// Mitsubishi GX Works2 project: PLC- Group36   PLC: FX3G

// global labels: Global1
VAR_GLOBAL
  Start AT X007 : BOOL;
  M_Cream AT D1100 : INT;
END_VAR
VAR_GLOBAL CONSTANT
  Min_Cream : INT := 300;
END_VAR
VAR_GLOBAL
  M_Chocolate AT D1200 : INT;
END_VAR
VAR_GLOBAL CONSTANT
  Min_Chocolate : INT := 240;
END_VAR
VAR_GLOBAL
  M_Bisc AT D1300 : INT;
END_VAR
VAR_GLOBAL CONSTANT
  Min_Bisc : INT := 6;
END_VAR
VAR_GLOBAL
  Lamp_Start AT Y007 : BOOL;
  KJK AT Y005 : BOOL;
  Start2 AT X010 : BOOL;
  Start_Cream AT X011 : BOOL;
END_VAR
VAR_GLOBAL CONSTANT
  Less_Cream : INT := 300;
  Less_Bisc : INT := 6;
END_VAR
VAR_GLOBAL
  Start_Dipping AT X006 : BOOL;
  Analog_Input1 AT D8280 : INT;
  Save_analog1 AT D8201 : INT;
  SaveLampInput AT M1 : BOOL;
END_VAR
VAR_GLOBAL CONSTANT
  Min_Analog1 : INT := 6;
  Max_Analog1 : INT := 5;
  Less_ChocolateA : INT := 240;
  Less_ChocolateB : INT := 120;
END_VAR
VAR_GLOBAL
  Timer_Dipping AT TC10 : BOOL;
END_VAR
VAR_GLOBAL CONSTANT
  Time_Value : INT := 50;
END_VAR
VAR_GLOBAL
  Lamp_Dipping AT Y003 : BOOL;
END_VAR
VAR_GLOBAL CONSTANT
  Div_Analog1 : INT := 400;
END_VAR
VAR_GLOBAL
  Time_1 AT TS10 : BOOL;
  check AT X000 : BOOL;
  Input_Cream AT D1110 : INT;
  Input_Bisc AT D1310 : INT;
  Input_Chocolate AT D1210 : INT;
  Time_10 AT M10 : BOOL;
  Timer_Moving AT TC2 : BOOL;
  Time_Value2 AT K10 : INT;
  Time_2 AT TS2 : BOOL;
  Moving_Lamp0 AT Y000 : BOOL;
  Timer_Moving2 AT TC3 : BOOL;
  Time_Value3 AT K10 : INT;
  Time_3 AT TS3 : BOOL;
  Moving_Lamp1 AT Y001 : BOOL;
  Timer_Moving3 AT TC4 : BOOL;
END_VAR
VAR_GLOBAL CONSTANT
  Time_Value4 : INT := K40;
END_VAR
VAR_GLOBAL
  Time_4 AT TS4 : BOOL;
  Start_wrrap AT X000 : BOOL;
  Counter_1 AT CC0 : BOOL;
  Counter_Value1 AT K5 : INT;
  Wrap_Light AT Y002 : BOOL;
  Count0 AT CS0 : BOOL;
  Counter_2 AT CC1 : BOOL;
  Counter_Value2 AT K6 : INT;
  Count_2 AT CS1 : BOOL;
  Start_A AT X010 : BOOL;
  System_A_On AT M0 : BOOL;
  Close_System_A AT X005 : BOOL;
  Sensor_Arrival AT X002 : BOOL;
  Camera_All AT X001 : BOOL;
  Sensor_30 AT X003 : BOOL;
  Sensor_15 AT X004 : BOOL;
  Machine_A_On AT Y004 : BOOL;
  Cont_Cream AT D1120 : INT;
  Cont_Choco AT D1220 : INT;
END_VAR
VAR_GLOBAL CONSTANT
  Decimal_Bisc : INT := 10;
END_VAR
VAR_GLOBAL
  Analon_Output AT D8282 : INT;
  End_A AT M6 : BOOL;
  EndOfDay AT M3 : BOOL;
  Timer_End5 AT TC5 : BOOL;
END_VAR
VAR_GLOBAL CONSTANT
  Time_Value5 : INT := K30;
END_VAR
VAR_GLOBAL
  Time_5 AT TS5 : BOOL;
  Time_End2 AT TC6 : BOOL;
END_VAR
VAR_GLOBAL CONSTANT
  Time_Value6 : INT := K5;
END_VAR
VAR_GLOBAL
  Time6 AT TS6 : BOOL;
  Lamp_Start1 AT Y011 : BOOL;
  Lamp_Start_Fake AT M7 : BOOL;
  Lamp_Fake AT M4 : BOOL;
  Time_End3 AT TC7 : BOOL;
  Time7 AT TS7 : BOOL;
  Time_11 AT M11 : BOOL;
  Fake_Lamp2 AT M20 : BOOL;
  Fake_Lamp3 AT M23 : BOOL;
END_VAR
VAR_GLOBAL CONSTANT
  Normalized_BiscNum : REAL := E6;
  Div_Analog2 : REAL := E40.0;
END_VAR
VAR_GLOBAL
  Num_Of_Krembo AT D1400 : REAL;
  Analog_Output AT D8282 : INT;
  Number_Bisc AT D1333 : REAL;
  Normal_Dip AT M15 : BOOL;
  Double_Dip AT M12 : BOOL;
  Stop_Dipping AT M13 : BOOL;
  Fin_Dip AT M14 : BOOL;
  Time_50 AT M50 : BOOL;
  Count_Lamp AT M34 : BOOL;
END_VAR

// task Task_01 (event TRUE, interval 0, priority 31): POU_01

PROGRAM POU_01
(* structured ladder/FBD written out as ST: instructions are called as NAME(EN, inputs, outputs); _pN, _eN, _tN stand for wires *)
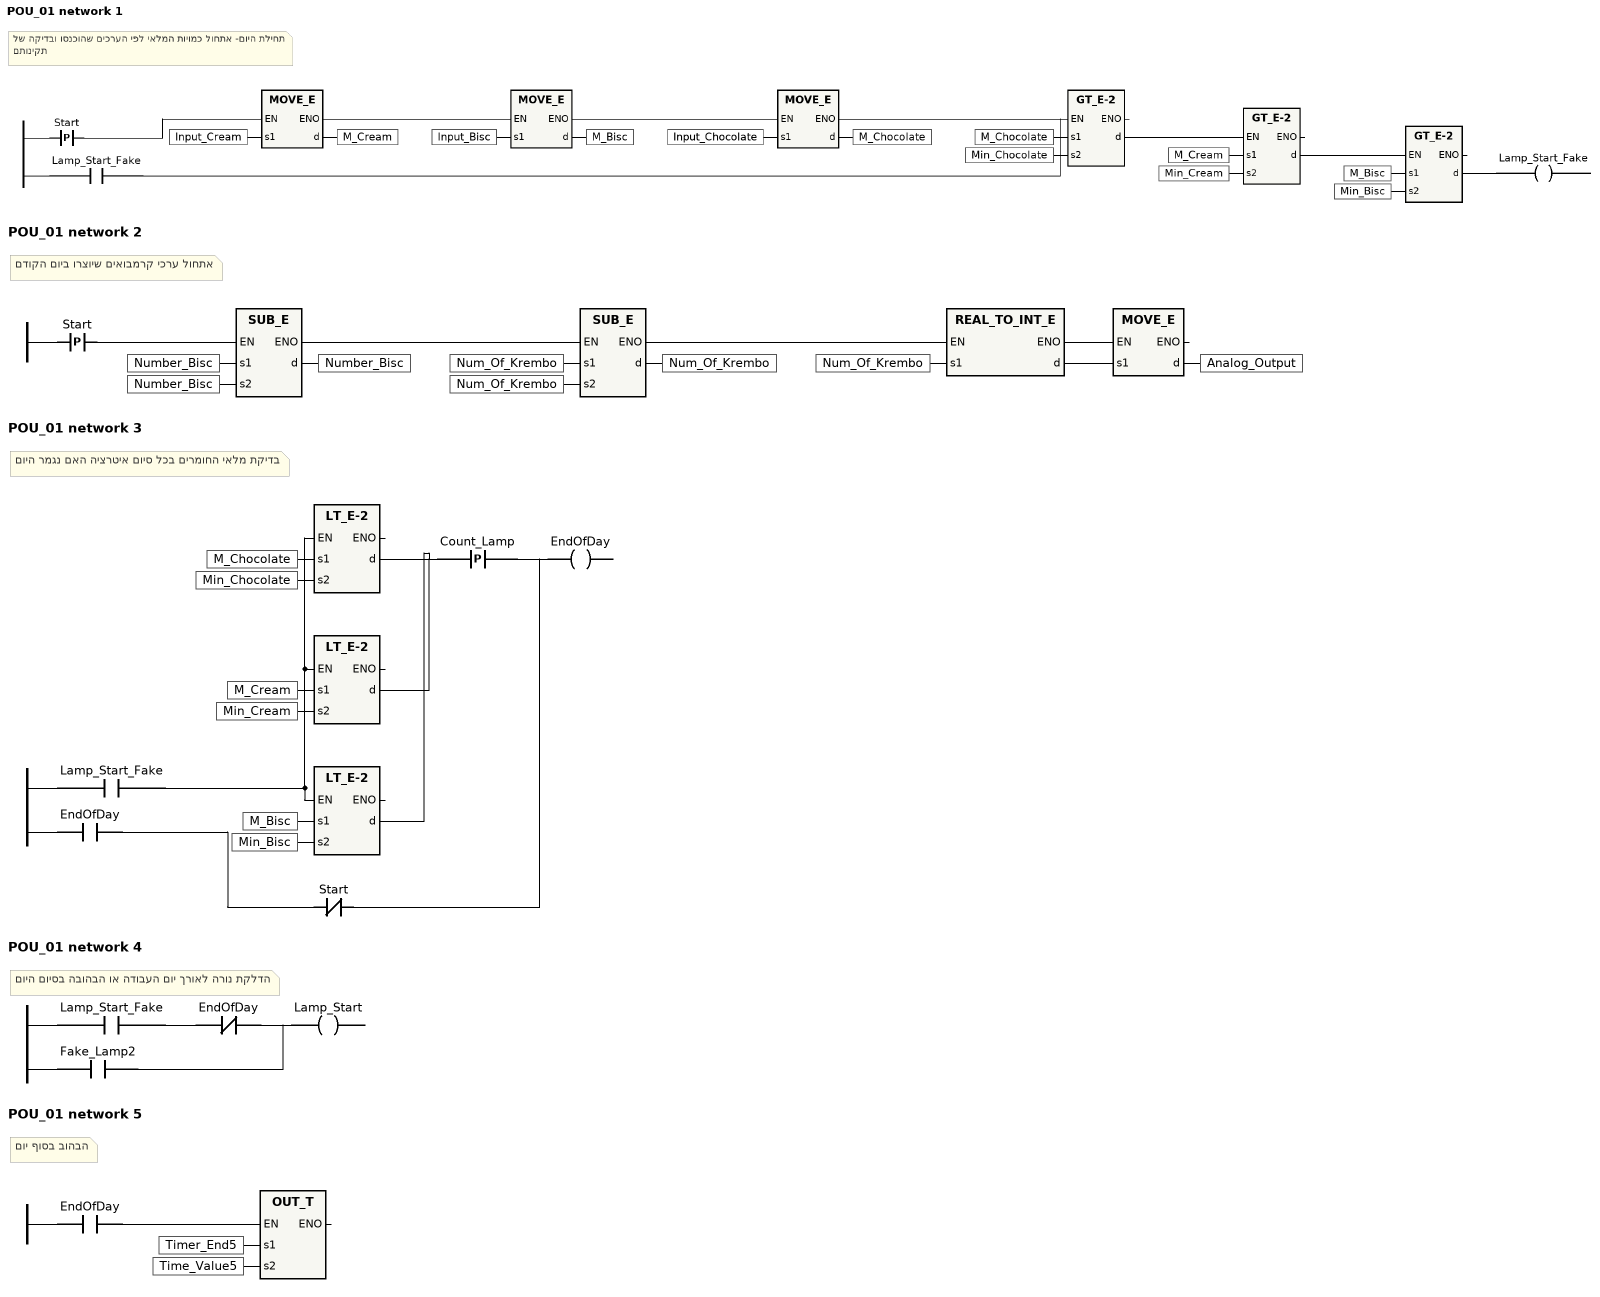
(* network 1 *)
(* תחילת היום- אתחול כמויות המלאי לפי הערכים שהוכנסו ובדיקה של תקינותם *)
_e1 := MOVE_E(LDP(TRUE, Start), Input_Cream, M_Cream);
_e2 := MOVE_E(_e1, Input_Bisc, M_Bisc);
_e3 := MOVE_E(_e2, Input_Chocolate, M_Chocolate);
GT_E(_e3 OR Lamp_Start_Fake, M_Chocolate, Min_Chocolate, _t4);
GT_E(_t4, M_Cream, Min_Cream, _t5);
GT_E(_t5, M_Bisc, Min_Bisc, _t6);
Lamp_Start_Fake := _t6;
(* network 2 *)
(* אתחול ערכי קרמבואים שיוצרו ביום הקודם *)
_e1 := SUB_E(LDP(TRUE, Start), Number_Bisc, Number_Bisc, Number_Bisc);
_e2 := SUB_E(_e1, Num_Of_Krembo, Num_Of_Krembo, Num_Of_Krembo);
_e4 := REAL_TO_INT_E(_e2, Num_Of_Krembo, _t3);
MOVE_E(_e4, _t3, Analog_Output);
(* network 3 *)
(* בדיקת מלאי החומרים בכל סיום איטרציה האם נגמר היום *)
LT_E(Lamp_Start_Fake, M_Chocolate, Min_Chocolate, _t1);
LT_E(Lamp_Start_Fake, M_Cream, Min_Cream, _t2);
LT_E(Lamp_Start_Fake, M_Bisc, Min_Bisc, _t3);
EndOfDay := ((_t1 OR _t2 OR _t3) AND LDP(TRUE, Count_Lamp)) OR (EndOfDay AND NOT Start);
(* network 4 *)
(* הדלקת נורה לאורך יום העבודה או הבהובה בסיום היום *)
Lamp_Start := (Lamp_Start_Fake AND NOT EndOfDay) OR Fake_Lamp2;
(* network 5 *)
(* הבהוב בסוף יום *)
OUT_T(EndOfDay, Timer_End5, Time_Value5);
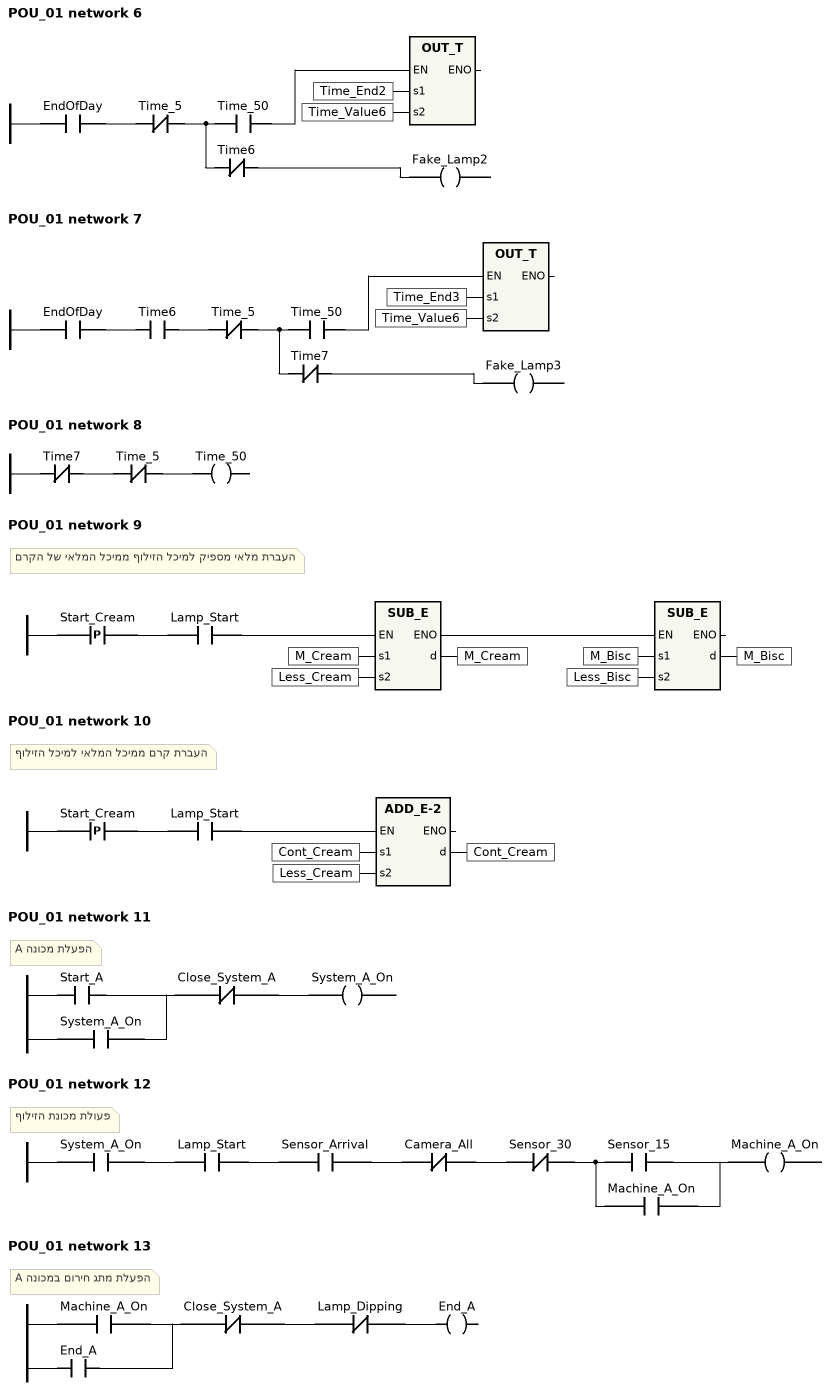
(* network 6 *)
_p1 := EndOfDay AND NOT Time_5;
OUT_T(_p1 AND Time_50, Time_End2, Time_Value6);
Fake_Lamp2 := _p1 AND NOT Time6;
(* network 7 *)
_p1 := EndOfDay AND Time6 AND NOT Time_5;
OUT_T(_p1 AND Time_50, Time_End3, Time_Value6);
Fake_Lamp3 := _p1 AND NOT Time7;
(* network 8 *)
Time_50 := NOT Time7 AND NOT Time_5;
(* network 9 *)
(* העברת מלאי מספיק למיכל הזילוף ממיכל המלאי של הקרם *)
_e1 := SUB_E(LDP(TRUE, Start_Cream) AND Lamp_Start, M_Cream, Less_Cream, M_Cream);
SUB_E(_e1, M_Bisc, Less_Bisc, M_Bisc);
(* network 10 *)
(* העברת קרם ממיכל המלאי למיכל הזילוף *)
ADD_E(LDP(TRUE, Start_Cream) AND Lamp_Start, Cont_Cream, Less_Cream, Cont_Cream);
(* network 11 *)
(* הפעלת מכונה A *)
System_A_On := (Start_A OR System_A_On) AND NOT Close_System_A;
(* network 12 *)
(* פעולת מכונת הזילוף *)
_p1 := System_A_On AND Lamp_Start AND Sensor_Arrival AND NOT Camera_All AND NOT Sensor_30;
Machine_A_On := (_p1 AND Sensor_15) OR (_p1 AND Machine_A_On);
(* network 13 *)
(* הפעלת מתג חירום במכונה A *)
End_A := ((Machine_A_On OR End_A) AND NOT Close_System_A) AND NOT Lamp_Dipping;
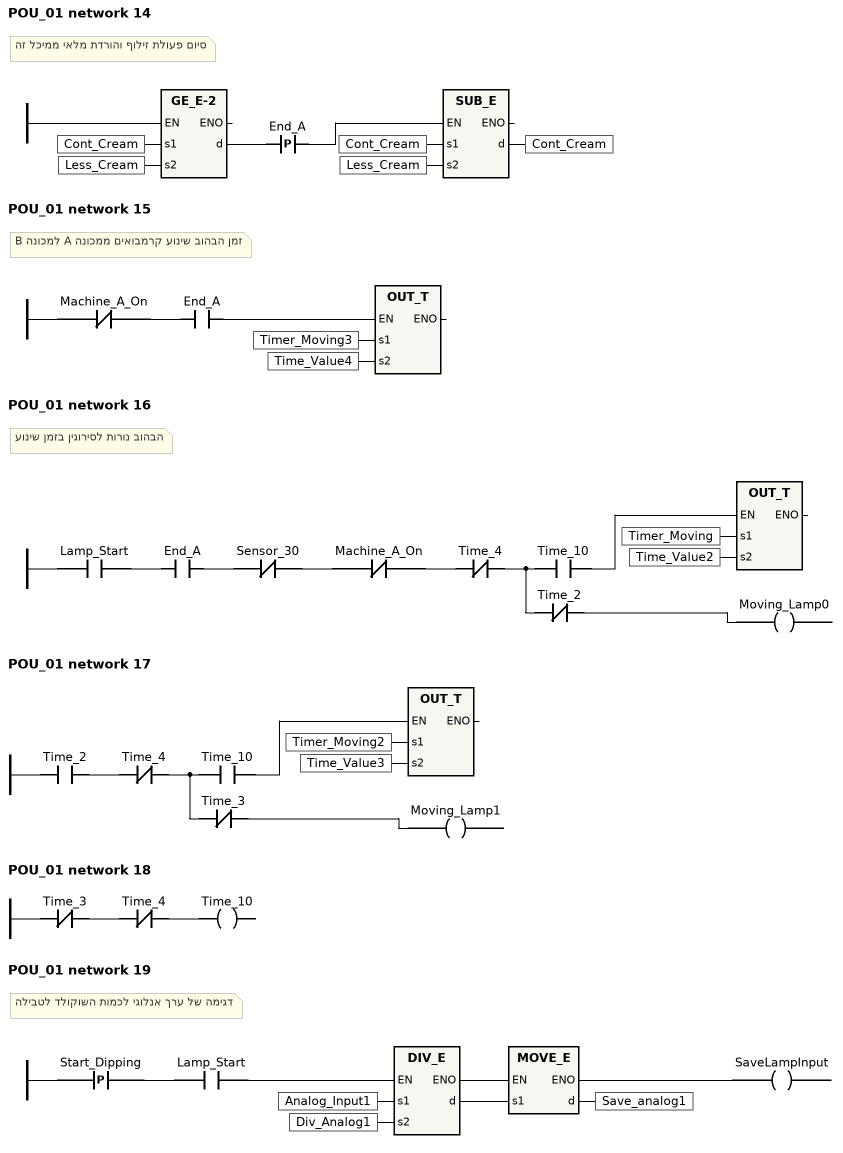
(* network 14 *)
(* סיום פעולת זילוף והורדת מלאי ממיכל זה *)
GE_E(TRUE, Cont_Cream, Less_Cream, _t1);
SUB_E(_t1 AND LDP(TRUE, End_A), Cont_Cream, Less_Cream, Cont_Cream);
(* network 15 *)
(* זמן הבהוב שינוע קרמבואים ממכונה A למכונה B *)
OUT_T(NOT Machine_A_On AND End_A, Timer_Moving3, Time_Value4);
(* network 16 *)
(* הבהוב נורות לסירוגין בזמן שינוע *)
_p1 := Lamp_Start AND End_A AND NOT Sensor_30 AND NOT Machine_A_On AND NOT Time_4;
OUT_T(_p1 AND Time_10, Timer_Moving, Time_Value2);
Moving_Lamp0 := _p1 AND NOT Time_2;
(* network 17 *)
_p1 := Time_2 AND NOT Time_4;
OUT_T(_p1 AND Time_10, Timer_Moving2, Time_Value3);
Moving_Lamp1 := _p1 AND NOT Time_3;
(* network 18 *)
Time_10 := NOT Time_3 AND NOT Time_4;
(* network 19 *)
(* דגימה של ערך אנלוגי לכמות השוקולד לטבילה *)
_e2 := DIV_E(LDP(TRUE, Start_Dipping) AND Lamp_Start, Analog_Input1, Div_Analog1, _t1);
_e3 := MOVE_E(_e2, _t1, Save_analog1);
SaveLampInput := _e3;
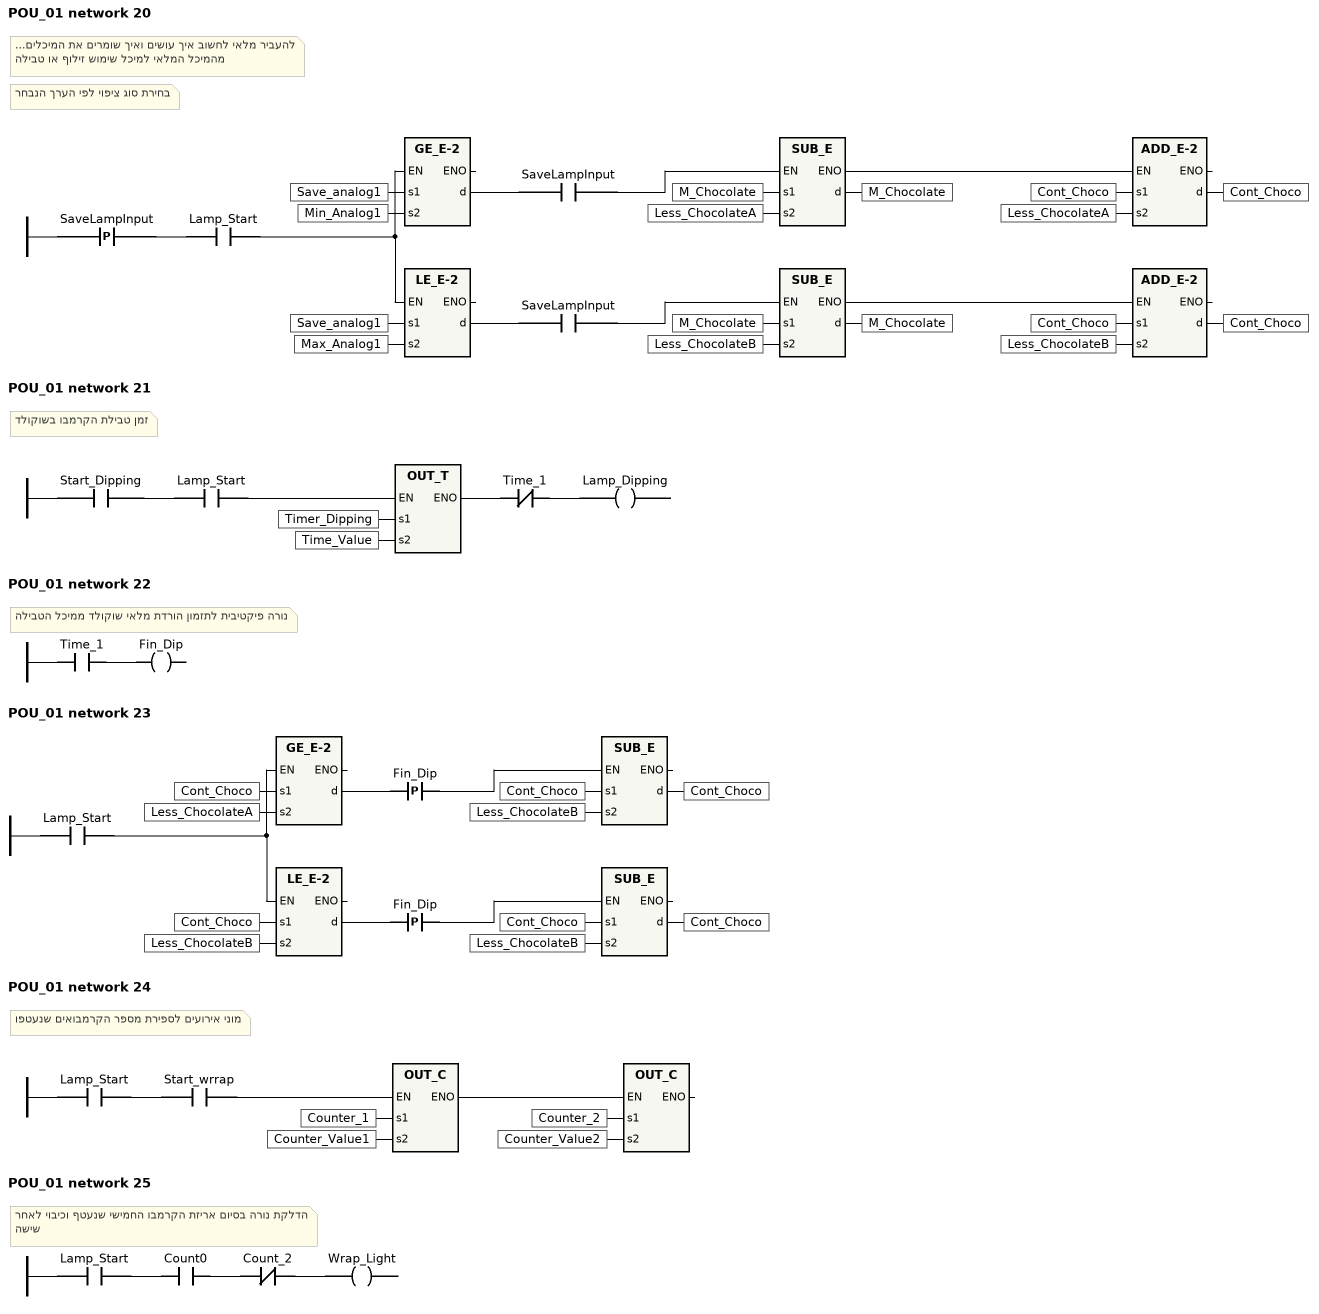
(* network 20 *)
(* להעביר מלאי לחשוב איך עושים ואיך שומרים את המיכלים... מהמיכל המלאי למיכל שימוש זילוף או טבילה *)
(* בחירת סוג ציפוי לפי הערך הנבחר *)
_p1 := LDP(TRUE, SaveLampInput) AND Lamp_Start;
GE_E(_p1, Save_analog1, Min_Analog1, _t2);
_e3 := SUB_E(_t2 AND SaveLampInput, M_Chocolate, Less_ChocolateA, M_Chocolate);
ADD_E(_e3, Cont_Choco, Less_ChocolateA, Cont_Choco);
LE_E(_p1, Save_analog1, Max_Analog1, _t4);
_e5 := SUB_E(_t4 AND SaveLampInput, M_Chocolate, Less_ChocolateB, M_Chocolate);
ADD_E(_e5, Cont_Choco, Less_ChocolateB, Cont_Choco);
(* network 21 *)
(* זמן טבילת הקרמבו בשוקולד *)
_e1 := OUT_T(Start_Dipping AND Lamp_Start, Timer_Dipping, Time_Value);
Lamp_Dipping := _e1 AND NOT Time_1;
(* network 22 *)
(* נורה פיקטיבית לתזמון הורדת מלאי שוקולד ממיכל הטבילה *)
Fin_Dip := Time_1;
(* network 23 *)
GE_E(Lamp_Start, Cont_Choco, Less_ChocolateA, _t1);
SUB_E(_t1 AND LDP(TRUE, Fin_Dip), Cont_Choco, Less_ChocolateB, Cont_Choco);
LE_E(Lamp_Start, Cont_Choco, Less_ChocolateB, _t2);
SUB_E(_t2 AND LDP(TRUE, Fin_Dip), Cont_Choco, Less_ChocolateB, Cont_Choco);
(* network 24 *)
(* מוני אירועים לספירת מספר הקרמבואים שנעטפו *)
_e1 := OUT_C(Lamp_Start AND Start_wrrap, Counter_1, Counter_Value1);
OUT_C(_e1, Counter_2, Counter_Value2);
(* network 25 *)
(* הדלקת נורה בסיום אריזת הקרמבו החמישי שנעטף וכיבוי לאחר שישה *)
Wrap_Light := Lamp_Start AND Count0 AND NOT Count_2;
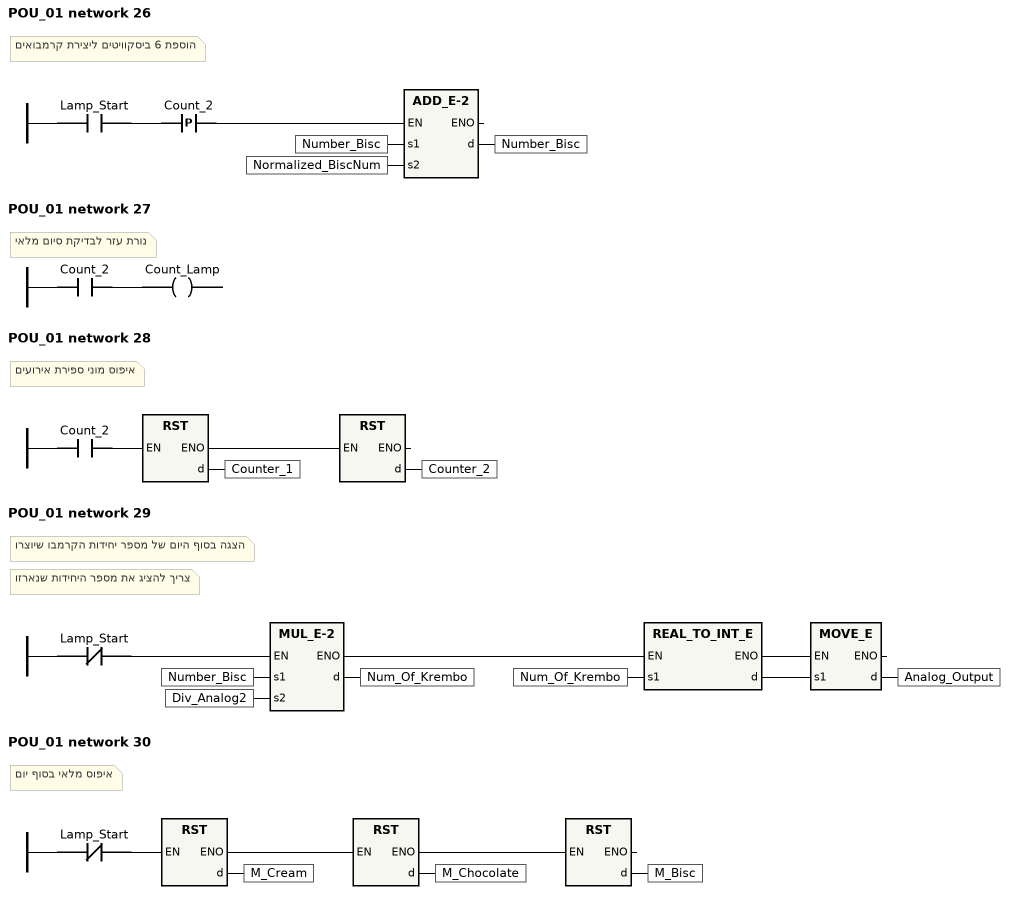
(* network 26 *)
(* הוספת 6 ביסקוויטים ליצירת קרמבואים *)
ADD_E(Lamp_Start AND LDP(TRUE, Count_2), Number_Bisc, Normalized_BiscNum, Number_Bisc);
(* network 27 *)
(* נורת עזר לבדיקת סיום מלאי *)
Count_Lamp := Count_2;
(* network 28 *)
(* איפוס מוני ספירת אירועים *)
_e1 := RST(Count_2, Counter_1);
RST(_e1, Counter_2);
(* network 29 *)
(* הצגה בסוף היום של מספר יחידות הקרמבו שיוצרו *)
(* צריך להציג את מספר היחידות שנארזו *)
_e1 := MUL_E(NOT Lamp_Start, Number_Bisc, Div_Analog2, Num_Of_Krembo);
_e3 := REAL_TO_INT_E(_e1, Num_Of_Krembo, _t2);
MOVE_E(_e3, _t2, Analog_Output);
(* network 30 *)
(* איפוס מלאי בסוף יום *)
_e1 := RST(NOT Lamp_Start, M_Cream);
_e2 := RST(_e1, M_Chocolate);
RST(_e2, M_Bisc);
END_PROGRAM
